// TIA Portal V17 export
// export: Created 2022-12-08T10:17:24.4855331Z, ExportSetting WithDefaults, DisplayName Totally Integrated Automation Portal, DisplayVersion V17 Update 5, DisplayName TIA Portal Openness, DisplayVersion V17 Update 5, DisplayName TIA Portal Version Control Interface, DisplayVersion V17, DisplayName Simotion SCOUT TIA, DisplayVersion 5.4.3.0, DisplayName SINAMICS Startdrive Advanced, DisplayVersion V17 SP1, DisplayName SINAMICS Startdrive G130, G150, S120, S150, SINAMICS MV, S210, DisplayVersion V17 SP1, DisplayName SINAMICS Startdrive G110M, G120, G120C, G120D, G120P, G115D, DisplayVersion V17 SP1, DisplayName STEP 7 Professional, DisplayVersion V17 Update 5, DisplayName STEP 7 Safety, DisplayVersion V17, DisplayName WinCC Advanced, DisplayVersion V17 Update 5
DATA_BLOCK "DB_UserManagement"   // DB28
VERSION : 0.1
// stored: AutoNumber true, DBAccessibleFromOPCUA true, DBAccessibleFromWebserver true, InstanceOfName FB_UserManagement, InstanceOfType FB
"FB_UserManagement"
   // VAR_INPUT
   //    i_PictureNumber : Int;
   // END_VAR
   // VAR_OUTPUT
   //    q_ActiveUser : "UDT_UserManagement";
   //    q_NoUserFound : Bool;
   //    q_UserAlreadyAdded : Bool;
   //    q_NewUserAdded : Bool;
   //    q_UserDeleted : Bool;
   // END_VAR
   // VAR_IN_OUT
   //    iq_HMIUserManagement : "UDT_HMIUserManagement";
   //    iq_User : Array[0.."UPPERUSERNUMBER"] of "UDT_UserManagement";
   // END_VAR
   // VAR
   //    stat_FirstScan : Bool;
   //    stat_TONLogOff : TON_TIME;
   //    stat_TONNoUserFound { S7_SetPoint := 'True'} : TON_TIME;
   //    stat_TONUserAlreadyAdded { S7_SetPoint := 'True'} : TON_TIME;
   //    stat_TONNewUserAdded { S7_SetPoint := 'True'} : TON_TIME;
   //    stat_TONUserDeleted { S7_SetPoint := 'True'} : TON_TIME;
   //    stat_ActiveUser { S7_SetPoint := 'True'} : "UDT_UserManagement";
   //    stat_UserLevel { ExternalAccessible := 'False'; ExternalVisible := 'False'; ExternalWritable := 'False'} : Array[0..4] of "UDT_UserAuthorisation";
   //    stat_NoUserFound : Bool;
   //    stat_UserAlreadyAdded : Bool;
   //    stat_NewUserAdded : Bool;
   //    stat_UserDeleted : Bool;
   //    stat_OldPictureNumber : Int;
   // END_VAR
BEGIN
END_DATA_BLOCK
